INTERFACE I_UniversalSafety

METHOD MR_Abort : BOOL
VAR_INPUT
END_VAR
END_METHOD

METHOD MR_FirstCycle : BOOL
VAR_INPUT
END_VAR
END_METHOD

METHOD MR_Init : BOOL
VAR_INPUT
END_VAR
END_METHOD

METHOD MR_Reset : BOOL
VAR_INPUT
END_VAR
END_METHOD

END_INTERFACE

(* stored: Version 1.1.0.1, ProductVersion 3.1.4024.9
   Itf I_UniversalSafety: Id {55f8c65a-c4ce-4380-8680-ab46b7bafc4a}
   Method MR_Abort: Id {06b7d620-0f2a-4512-bf69-38cf69cc1707}
   Method MR_FirstCycle: Id {620dfdff-9a97-43f7-9a0b-16bdd9ffbd15}
   Method MR_Init: Id {2c729596-a4c8-4a74-a26e-93e599e95f8e}
   Method MR_Reset: Id {617cffb6-73de-46f9-a483-16d3a7382244} *)
